SUBAPPLICATION Uebung_012a_AX (* Numeric Value Input und Speichern (Adapter Version) *)
  (* Standard: 61499-2; Description: Copyright (c) 2026 Meisterschulen am Ostbahnhof This program and the accompanying materials are made available under the terms of the Eclipse Public License 2.0 which is available at https://www.eclipse.org/legal/epl-2.0/ SPDX-License-Identifier: EPL-2.0 *)
  (* Version 1.0, 2026-04-21, Franz Höpfinger, Meisterschulen am Ostbahnhof, initial API and implementation (AX version) *)
  PACKAGE Uebungen;
  IMPORT Uebungen::const::NVS::NVS_Keys::KEY_I1_STORE;
  IMPORT Uebungen::const::UT::DefaultPool::InputNumber_I1;
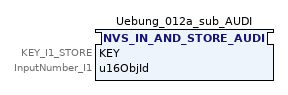
  SUBAPPS
    Uebung_012a_sub_AUDI : MyLib::sys::NVS_IN_AND_STORE_AUDI(KEY := KEY_I1_STORE, u16ObjId := InputNumber_I1);
  END_SUBAPPS
END_SUBAPPLICATION
